// TIA Portal V16 export
// export: Created 2021-06-11T05:47:00.3145805Z, ExportSetting WithDefaults, DisplayName Totally Integrated Automation Portal, DisplayVersion V16 Update 4, DisplayName TIA Portal Version Control Interface, DisplayVersion V16 Update 2, DisplayName TIA Portal Openness, DisplayVersion V16 Update 4, DisplayName TIA Portal Teamcenter Gateway, DisplayVersion V16, DisplayName SINAMICS Startdrive Advanced, DisplayVersion V16 Update 5, DisplayName SINAMICS Startdrive G130, G150, S120, S150, SINAMICS MV, S210, DisplayVersion V16 Update 5, DisplayName SINAMICS Startdrive G110M, G120, G120C, G120D, G120P, G115D, DisplayVersion V16 Update 5, DisplayName STEP 7 Professional, DisplayVersion V16 Update 4, DisplayName SINUMERIK ONE STEP 7 Toolbox, DisplayVersion V16 Update 3, DisplayName STEP 7 Safety, DisplayVersion V16, DisplayName SINUMERIK 840D sl STEP 7 Toolbox, DisplayVersion V16 Update 2, DisplayName WinCC Advanced, DisplayVersion V16 Update 4
FUNCTION "FC_OperatingModes" : Void   // FC1601, LAD
{ S7_Optimized_Access := 'TRUE' }
VERSION : 0.1
// stored: AutoNumber false, IsIECCheckEnabled false, SetENOAutomatically true, UDAEnableTagReadback false
   VAR_TEMP
      tx_OperatingMode_KeyDisable : Bool;
      tb_DialogEnable : Byte;
      tx_DialogEnable : Array[0..7] of Bool;
      tint_Ret_Val : Int;
      WcsMcs_Edge : Bool;
      WcsMcs_Flag : Bool;
   END_VAR
BEGIN

REGION Network 1: MCP
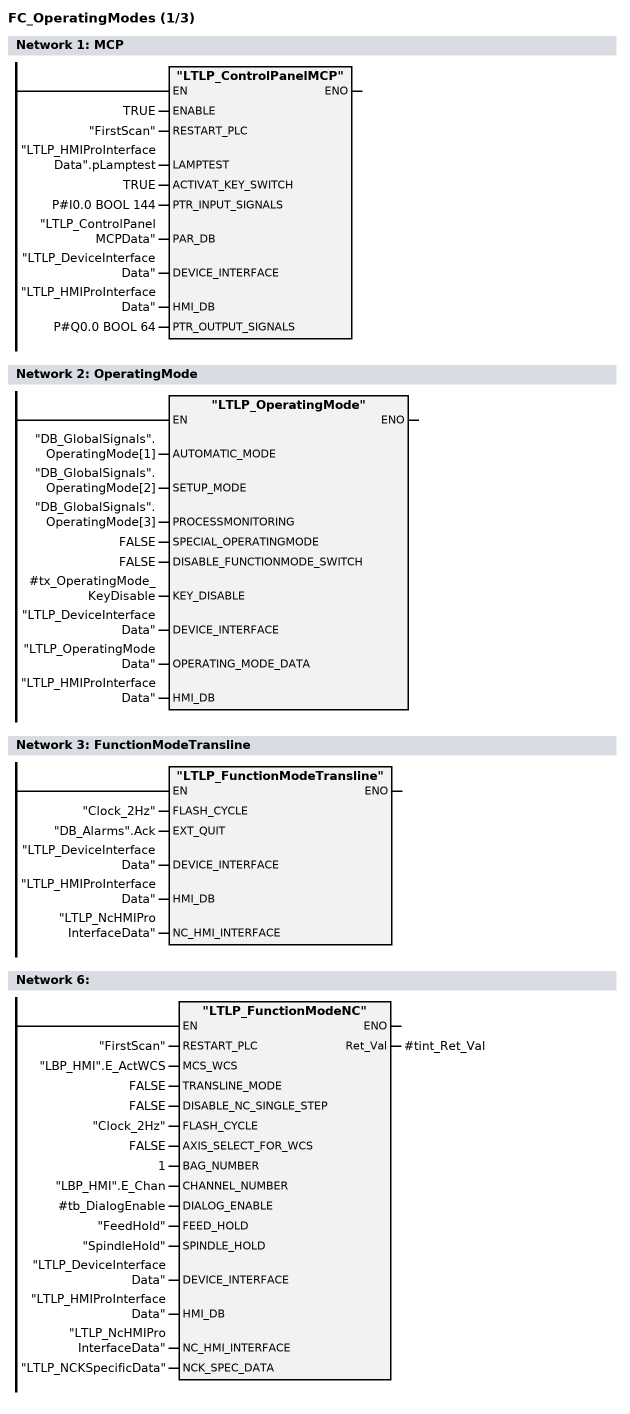
   RUNG wire#powerrail
      "LTLP_ControlPanelMCP"(ENABLE := TRUE, RESTART_PLC := "FirstScan", LAMPTEST := "LTLP_HMIProInterfaceData".pLamptest, ACTIVAT_KEY_SWITCH := TRUE, PTR_INPUT_SIGNALS := P#I0.0 BOOL 144, PAR_DB := "LTLP_ControlPanelMCPData", DEVICE_INTERFACE := "LTLP_DeviceInterfaceData", HMI_DB := "LTLP_HMIProInterfaceData", PTR_OUTPUT_SIGNALS := P#Q0.0 BOOL 64)
   END_RUNG
   // the same network as SCL:
   "LTLP_ControlPanelMCP"(ENABLE := TRUE,
                          RESTART_PLC := "FirstScan",
                          LAMPTEST := "LTLP_HMIProInterfaceData".pLamptest,
                          ACTIVAT_KEY_SWITCH := TRUE,
                          PTR_INPUT_SIGNALS := P#I0.0 BOOL 144,
                          PAR_DB := "LTLP_ControlPanelMCPData",
                          DEVICE_INTERFACE := "LTLP_DeviceInterfaceData",
                          HMI_DB := "LTLP_HMIProInterfaceData",
                          PTR_OUTPUT_SIGNALS := P#Q0.0 BOOL 64);
END_REGION

REGION Network 2: OperatingMode
   RUNG wire#powerrail
      "LTLP_OperatingMode"(AUTOMATIC_MODE := "DB_GlobalSignals".OperatingMode[1], SETUP_MODE := "DB_GlobalSignals".OperatingMode[2], PROCESSMONITORING := "DB_GlobalSignals".OperatingMode[3], SPECIAL_OPERATINGMODE := FALSE, DISABLE_FUNCTIONMODE_SWITCH := FALSE, KEY_DISABLE := #tx_OperatingMode_KeyDisable, DEVICE_INTERFACE := "LTLP_DeviceInterfaceData", OPERATING_MODE_DATA := "LTLP_OperatingModeData", HMI_DB := "LTLP_HMIProInterfaceData")
   END_RUNG
   // the same network as SCL:
   "LTLP_OperatingMode"(AUTOMATIC_MODE := "DB_GlobalSignals".OperatingMode[1],
                        SETUP_MODE := "DB_GlobalSignals".OperatingMode[2],
                        PROCESSMONITORING := "DB_GlobalSignals".OperatingMode[3],
                        SPECIAL_OPERATINGMODE := FALSE,
                        DISABLE_FUNCTIONMODE_SWITCH := FALSE,
                        KEY_DISABLE := #tx_OperatingMode_KeyDisable,
                        DEVICE_INTERFACE := "LTLP_DeviceInterfaceData",
                        OPERATING_MODE_DATA := "LTLP_OperatingModeData",
                        HMI_DB := "LTLP_HMIProInterfaceData");
END_REGION

REGION Network 3: FunctionModeTransline
   RUNG wire#powerrail
      "LTLP_FunctionModeTransline"(FLASH_CYCLE := "Clock_2Hz", EXT_QUIT := "DB_Alarms".Ack, DEVICE_INTERFACE := "LTLP_DeviceInterfaceData", HMI_DB := "LTLP_HMIProInterfaceData", NC_HMI_INTERFACE := "LTLP_NcHMIProInterfaceData")
   END_RUNG
   // the same network as SCL:
   "LTLP_FunctionModeTransline"(FLASH_CYCLE := "Clock_2Hz",
                           EXT_QUIT := "DB_Alarms".Ack,
                           DEVICE_INTERFACE := "LTLP_DeviceInterfaceData",
                           HMI_DB := "LTLP_HMIProInterfaceData",
                           NC_HMI_INTERFACE := "LTLP_NcHMIProInterfaceData");
END_REGION

REGION Network 4 (SCL)
   #tx_DialogEnable[0] := TRUE;
   #tx_DialogEnable[1] := TRUE;
   #tx_DialogEnable[2] := TRUE;
   #tx_DialogEnable[3] := FALSE;
   #tx_DialogEnable[4] := FALSE;
   #tx_DialogEnable[5] := FALSE;
   #tx_DialogEnable[6] := FALSE;
   #tx_DialogEnable[7] := TRUE;

   GATHER(IN := #tx_DialogEnable,
          OUT => #tb_DialogEnable);

   "LTLP_NCKSpecificData".Common.maxBAG := "LBP_ConfigData".MaxModeGroup;
   "LTLP_NCKSpecificData".Common.maxChannels := "LBP_ConfigData".MaxChan;
   "LTLP_NCKSpecificData".Common.maxAxis := "LBP_ConfigData".MaxAxis;

   "LTLP_NCKSpecificData".NCK.A_incInModeGroup := "LBP_NC".A_IncInModeGroup;
   "LTLP_NCKSpecificData".MMC.activeChannel := "LBP_HMI".E_Chan;

   //Flanke - System betriebsbereit
   "IDB_R_TRIG_SystemReady"(CLK := "LBP_NC".E_NCKready AND "LBP_NC".E_NCready AND "LBP_NC".E_DrivesInCylOp);

   //FeedStart im Hochlauf setzen
   IF "IDB_R_TRIG_SystemReady".Q THEN
       "LTLP_DeviceInterfaceData".inputs.mcpFunctions.feedStart := TRUE;
   ELSIF NOT "FeedHold" THEN
       "LTLP_DeviceInterfaceData".inputs.mcpFunctions.feedStart := FALSE;
   END_IF;
   //SpindleStart im Hochlauf setzen
   IF "IDB_R_TRIG_SystemReady".Q THEN
       "LTLP_DeviceInterfaceData".inputs.mcpFunctions.spindleStart := TRUE;
   ELSIF NOT "SpindleHold" THEN
       "LTLP_DeviceInterfaceData".inputs.mcpFunctions.spindleStart := FALSE;
   END_IF;
END_REGION

REGION Network 5 (SCL): bagDataSpecification
   // BAG
   "LTLP_NcHMIProInterfaceData".bagDataFeedback.auto := "LBP_ModeGroup".E_AUTO;
   "LTLP_NcHMIProInterfaceData".bagDataFeedback.mda := "LBP_ModeGroup".E_MDA;
   "LTLP_NcHMIProInterfaceData".bagDataFeedback.jog := "LBP_ModeGroup".E_JOG;
   "LTLP_NcHMIProInterfaceData".bagDataFeedback.inrement1 := "LBP_ModeGroup".E_INC1;
   "LTLP_NcHMIProInterfaceData".bagDataFeedback.inrement10 := "LBP_ModeGroup".E_INC10;
   "LTLP_NcHMIProInterfaceData".bagDataFeedback.inrement100 := "LBP_ModeGroup".E_INC100;
   "LTLP_NcHMIProInterfaceData".bagDataFeedback.increment1000 := "LBP_ModeGroup".E_INC1000;
   "LTLP_NcHMIProInterfaceData".bagDataFeedback.increment10000 := "LBP_ModeGroup".E_INC10000;
   "LTLP_NcHMIProInterfaceData".bagDataFeedback.incremetVariable := "LBP_ModeGroup".E_INCVar;
   "LTLP_NcHMIProInterfaceData".bagDataFeedback.gotoRefPoint := "LBP_ModeGroup".E_REF;
   "LTLP_NcHMIProInterfaceData".bagDataFeedback.teach := "LBP_ModeGroup".E_TEACHIN;

   // Channel
   "LTLP_NcHMIProInterfaceData".channelDataFeedback.rapidTraverse := "LTLP_DeviceInterfaceData".inputs.mcpFunctions.rapid;
   "LTLP_NcHMIProInterfaceData".channelDataFeedback.motionPlus := "LTLP_DeviceInterfaceData".inputs.mcpFunctions.motionPlus;
   "LTLP_NcHMIProInterfaceData".channelDataFeedback.motionMinus := "LTLP_DeviceInterfaceData".inputs.mcpFunctions.motionMinus;
   "LTLP_NcHMIProInterfaceData".channelDataFeedback.ncStart := "LTLP_DeviceInterfaceData".inputs.mcpFunctions.ncStart;
   "LTLP_NcHMIProInterfaceData".channelDataFeedback.ncStop := "LTLP_DeviceInterfaceData".inputs.mcpFunctions.ncStop;
   "LTLP_NcHMIProInterfaceData".channelDataFeedback.reset := "LTLP_DeviceInterfaceData".inputs.mcpFunctions.reset;
   "LTLP_NcHMIProInterfaceData".channelDataFeedback.singleBlock := "LBP_Chan1".A_SBL;

   // Axis
   "LTLP_NcHMIProInterfaceData".axisFeedback.rapidTraverse := "LTLP_DeviceInterfaceData".inputs.mcpFunctions.rapid;
   "LTLP_NcHMIProInterfaceData".axisFeedback.motionPlus := "LTLP_DeviceInterfaceData".inputs.mcpFunctions.motionPlus;
   "LTLP_NcHMIProInterfaceData".axisFeedback.motionMinus := "LTLP_DeviceInterfaceData".inputs.mcpFunctions.motionMinus;

   // Achse abwählen, falls AUTO oder MDA aktiv
   IF "LTLP_NcHMIProInterfaceData".bagDataFeedback.auto OR "LTLP_NcHMIProInterfaceData".bagDataFeedback.mda THEN
       "LTLP_NcHMIProInterfaceData".fromPlc.axisNoMcp := 0;
   END_IF;
END_REGION

REGION Network 6
   RUNG wire#powerrail
      "LTLP_FunctionModeNC"(RESTART_PLC := "FirstScan", MCS_WCS := "LBP_HMI".E_ActWCS, TRANSLINE_MODE := FALSE, DISABLE_NC_SINGLE_STEP := FALSE, FLASH_CYCLE := "Clock_2Hz", AXIS_SELECT_FOR_WCS := FALSE, BAG_NUMBER := 1, CHANNEL_NUMBER := "LBP_HMI".E_Chan, DIALOG_ENABLE := #tb_DialogEnable, FEED_HOLD := "FeedHold", SPINDLE_HOLD := "SpindleHold", DEVICE_INTERFACE := "LTLP_DeviceInterfaceData", HMI_DB := "LTLP_HMIProInterfaceData", NC_HMI_INTERFACE := "LTLP_NcHMIProInterfaceData", NCK_SPEC_DATA := "LTLP_NCKSpecificData", Ret_Val => #tint_Ret_Val)
   END_RUNG
   // the same network as SCL:
   #tint_Ret_Val := "LTLP_FunctionModeNC"(RESTART_PLC := "FirstScan",
                           MCS_WCS := "LBP_HMI".E_ActWCS,
                           TRANSLINE_MODE := FALSE,
                           DISABLE_NC_SINGLE_STEP := FALSE,
                           FLASH_CYCLE := "Clock_2Hz",
                           AXIS_SELECT_FOR_WCS := FALSE,
                           BAG_NUMBER := 1,
                           CHANNEL_NUMBER := "LBP_HMI".E_Chan,
                           DIALOG_ENABLE := #tb_DialogEnable,
                           FEED_HOLD := "FeedHold",
                           SPINDLE_HOLD := "SpindleHold",
                           DEVICE_INTERFACE := "LTLP_DeviceInterfaceData",
                           HMI_DB := "LTLP_HMIProInterfaceData",
                           NC_HMI_INTERFACE := "LTLP_NcHMIProInterfaceData",
                           NCK_SPEC_DATA := "LTLP_NCKSpecificData");
END_REGION

REGION Network 7: Betriebsarten
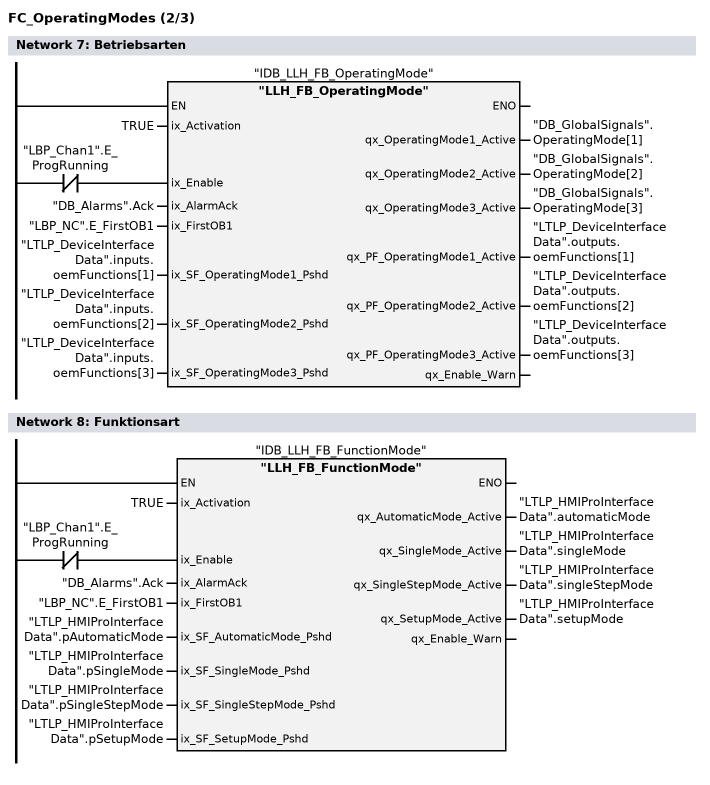
   RUNG wire#powerrail
      "IDB_LLH_FB_OperatingMode"(ix_Enable := wire#w1, ix_Activation := TRUE, ix_AlarmAck := "DB_Alarms".Ack, ix_FirstOB1 := "LBP_NC".E_FirstOB1, ix_SF_OperatingMode1_Pshd := "LTLP_DeviceInterfaceData".inputs.oemFunctions[1], ix_SF_OperatingMode2_Pshd := "LTLP_DeviceInterfaceData".inputs.oemFunctions[2], ix_SF_OperatingMode3_Pshd := "LTLP_DeviceInterfaceData".inputs.oemFunctions[3], qx_OperatingMode1_Active => "DB_GlobalSignals".OperatingMode[1], qx_OperatingMode2_Active => "DB_GlobalSignals".OperatingMode[2], qx_OperatingMode3_Active => "DB_GlobalSignals".OperatingMode[3], qx_PF_OperatingMode1_Active => "LTLP_DeviceInterfaceData".outputs.oemFunctions[1], qx_PF_OperatingMode2_Active => "LTLP_DeviceInterfaceData".outputs.oemFunctions[2], qx_PF_OperatingMode3_Active => "LTLP_DeviceInterfaceData".outputs.oemFunctions[3], qx_Enable_Warn =>)
   END_RUNG
   RUNG wire#powerrail
      I_Contact( "LBP_Chan1".E_ProgRunning )
   END_RUNG wire#w1
   // the same network as SCL:
   "IDB_LLH_FB_OperatingMode"(ix_Activation := TRUE,   // "LLH_FB_OperatingMode"
                           ix_Enable := NOT "LBP_Chan1".E_ProgRunning,
                           ix_AlarmAck := "DB_Alarms".Ack,
                           ix_FirstOB1 := "LBP_NC".E_FirstOB1,
                           ix_SF_OperatingMode1_Pshd := "LTLP_DeviceInterfaceData".inputs.oemFunctions[1],
                           ix_SF_OperatingMode2_Pshd := "LTLP_DeviceInterfaceData".inputs.oemFunctions[2],
                           ix_SF_OperatingMode3_Pshd := "LTLP_DeviceInterfaceData".inputs.oemFunctions[3],
                           qx_OperatingMode1_Active => "DB_GlobalSignals".OperatingMode[1],
                           qx_OperatingMode2_Active => "DB_GlobalSignals".OperatingMode[2],
                           qx_OperatingMode3_Active => "DB_GlobalSignals".OperatingMode[3],
                           qx_PF_OperatingMode1_Active => "LTLP_DeviceInterfaceData".outputs.oemFunctions[1],
                           qx_PF_OperatingMode2_Active => "LTLP_DeviceInterfaceData".outputs.oemFunctions[2],
                           qx_PF_OperatingMode3_Active => "LTLP_DeviceInterfaceData".outputs.oemFunctions[3]);
END_REGION

REGION Network 8: Funktionsart
   RUNG wire#powerrail
      "IDB_LLH_FB_FunctionMode"(ix_Enable := wire#w1, ix_Activation := TRUE, ix_AlarmAck := "DB_Alarms".Ack, ix_FirstOB1 := "LBP_NC".E_FirstOB1, ix_SF_AutomaticMode_Pshd := "LTLP_HMIProInterfaceData".pAutomaticMode, ix_SF_SingleMode_Pshd := "LTLP_HMIProInterfaceData".pSingleMode, ix_SF_SingleStepMode_Pshd := "LTLP_HMIProInterfaceData".pSingleStepMode, ix_SF_SetupMode_Pshd := "LTLP_HMIProInterfaceData".pSetupMode, qx_AutomaticMode_Active => "LTLP_HMIProInterfaceData".automaticMode, qx_SingleMode_Active => "LTLP_HMIProInterfaceData".singleMode, qx_SingleStepMode_Active => "LTLP_HMIProInterfaceData".singleStepMode, qx_SetupMode_Active => "LTLP_HMIProInterfaceData".setupMode, qx_Enable_Warn =>)
   END_RUNG
   RUNG wire#powerrail
      I_Contact( "LBP_Chan1".E_ProgRunning )
   END_RUNG wire#w1
   // the same network as SCL:
   "IDB_LLH_FB_FunctionMode"(ix_Activation := TRUE,   // "LLH_FB_FunctionMode"
                           ix_Enable := NOT "LBP_Chan1".E_ProgRunning,
                           ix_AlarmAck := "DB_Alarms".Ack,
                           ix_FirstOB1 := "LBP_NC".E_FirstOB1,
                           ix_SF_AutomaticMode_Pshd := "LTLP_HMIProInterfaceData".pAutomaticMode,
                           ix_SF_SingleMode_Pshd := "LTLP_HMIProInterfaceData".pSingleMode,
                           ix_SF_SingleStepMode_Pshd := "LTLP_HMIProInterfaceData".pSingleStepMode,
                           ix_SF_SetupMode_Pshd := "LTLP_HMIProInterfaceData".pSetupMode,
                           qx_AutomaticMode_Active => "LTLP_HMIProInterfaceData".automaticMode,
                           qx_SingleMode_Active => "LTLP_HMIProInterfaceData".singleMode,
                           qx_SingleStepMode_Active => "LTLP_HMIProInterfaceData".singleStepMode,
                           qx_SetupMode_Active => "LTLP_HMIProInterfaceData".setupMode);
END_REGION

REGION Network 9: ModeGroup
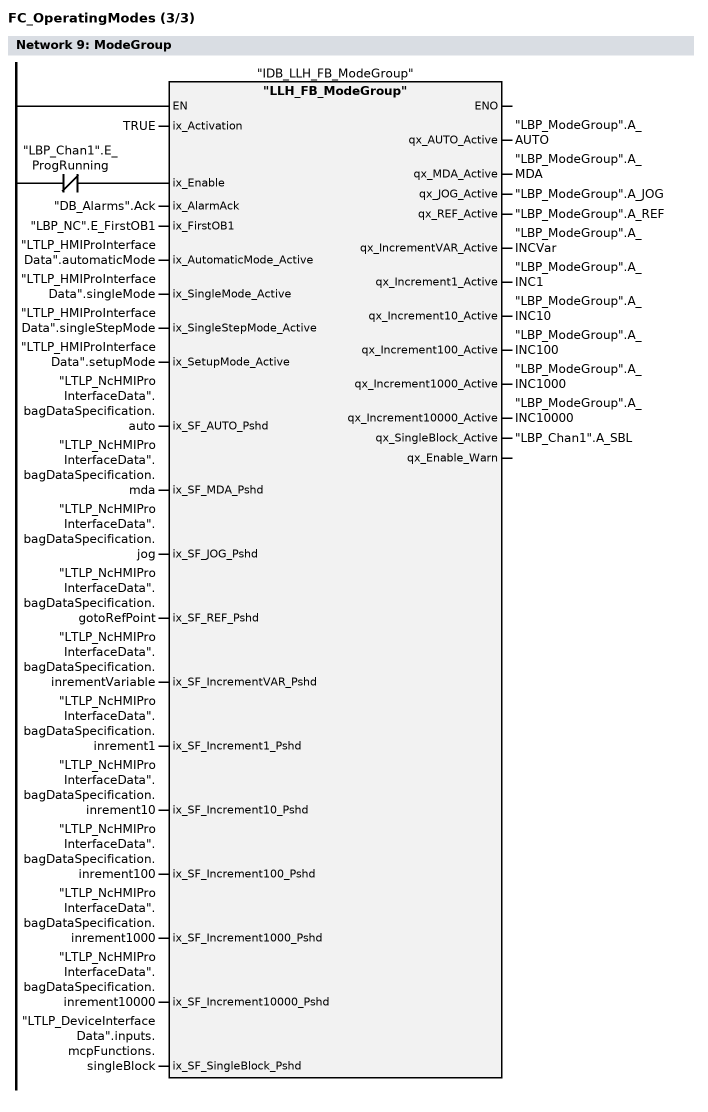
   RUNG wire#powerrail
      "IDB_LLH_FB_ModeGroup"(ix_Enable := wire#w1, ix_Activation := TRUE, ix_AlarmAck := "DB_Alarms".Ack, ix_FirstOB1 := "LBP_NC".E_FirstOB1, ix_AutomaticMode_Active := "LTLP_HMIProInterfaceData".automaticMode, ix_SingleMode_Active := "LTLP_HMIProInterfaceData".singleMode, ix_SingleStepMode_Active := "LTLP_HMIProInterfaceData".singleStepMode, ix_SetupMode_Active := "LTLP_HMIProInterfaceData".setupMode, ix_SF_AUTO_Pshd := "LTLP_NcHMIProInterfaceData".bagDataSpecification.auto, ix_SF_MDA_Pshd := "LTLP_NcHMIProInterfaceData".bagDataSpecification.mda, ix_SF_JOG_Pshd := "LTLP_NcHMIProInterfaceData".bagDataSpecification.jog, ix_SF_REF_Pshd := "LTLP_NcHMIProInterfaceData".bagDataSpecification.gotoRefPoint, ix_SF_IncrementVAR_Pshd := "LTLP_NcHMIProInterfaceData".bagDataSpecification.inrementVariable, ix_SF_Increment1_Pshd := "LTLP_NcHMIProInterfaceData".bagDataSpecification.inrement1, ix_SF_Increment10_Pshd := "LTLP_NcHMIProInterfaceData".bagDataSpecification.inrement10, ix_SF_Increment100_Pshd := "LTLP_NcHMIProInterfaceData".bagDataSpecification.inrement100, ix_SF_Increment1000_Pshd := "LTLP_NcHMIProInterfaceData".bagDataSpecification.inrement1000, ix_SF_Increment10000_Pshd := "LTLP_NcHMIProInterfaceData".bagDataSpecification.inrement10000, ix_SF_SingleBlock_Pshd := "LTLP_DeviceInterfaceData".inputs.mcpFunctions.singleBlock, qx_AUTO_Active => "LBP_ModeGroup".A_AUTO, qx_MDA_Active => "LBP_ModeGroup".A_MDA, qx_JOG_Active => "LBP_ModeGroup".A_JOG, qx_REF_Active => "LBP_ModeGroup".A_REF, qx_IncrementVAR_Active => "LBP_ModeGroup".A_INCVar, qx_Increment1_Active => "LBP_ModeGroup".A_INC1, qx_Increment10_Active => "LBP_ModeGroup".A_INC10, qx_Increment100_Active => "LBP_ModeGroup".A_INC100, qx_Increment1000_Active => "LBP_ModeGroup".A_INC1000, qx_Increment10000_Active => "LBP_ModeGroup".A_INC10000, qx_SingleBlock_Active => "LBP_Chan1".A_SBL, qx_Enable_Warn =>)
   END_RUNG
   RUNG wire#powerrail
      I_Contact( "LBP_Chan1".E_ProgRunning )
   END_RUNG wire#w1
   // the same network as SCL:
   "IDB_LLH_FB_ModeGroup"(ix_Activation := TRUE,   // "LLH_FB_ModeGroup"
                          ix_Enable := NOT "LBP_Chan1".E_ProgRunning,
                          ix_AlarmAck := "DB_Alarms".Ack,
                          ix_FirstOB1 := "LBP_NC".E_FirstOB1,
                          ix_AutomaticMode_Active := "LTLP_HMIProInterfaceData".automaticMode,
                          ix_SingleMode_Active := "LTLP_HMIProInterfaceData".singleMode,
                          ix_SingleStepMode_Active := "LTLP_HMIProInterfaceData".singleStepMode,
                          ix_SetupMode_Active := "LTLP_HMIProInterfaceData".setupMode,
                          ix_SF_AUTO_Pshd := "LTLP_NcHMIProInterfaceData".bagDataSpecification.auto,
                          ix_SF_MDA_Pshd := "LTLP_NcHMIProInterfaceData".bagDataSpecification.mda,
                          ix_SF_JOG_Pshd := "LTLP_NcHMIProInterfaceData".bagDataSpecification.jog,
                          ix_SF_REF_Pshd := "LTLP_NcHMIProInterfaceData".bagDataSpecification.gotoRefPoint,
                          ix_SF_IncrementVAR_Pshd := "LTLP_NcHMIProInterfaceData".bagDataSpecification.inrementVariable,
                          ix_SF_Increment1_Pshd := "LTLP_NcHMIProInterfaceData".bagDataSpecification.inrement1,
                          ix_SF_Increment10_Pshd := "LTLP_NcHMIProInterfaceData".bagDataSpecification.inrement10,
                          ix_SF_Increment100_Pshd := "LTLP_NcHMIProInterfaceData".bagDataSpecification.inrement100,
                          ix_SF_Increment1000_Pshd := "LTLP_NcHMIProInterfaceData".bagDataSpecification.inrement1000,
                          ix_SF_Increment10000_Pshd := "LTLP_NcHMIProInterfaceData".bagDataSpecification.inrement10000,
                          ix_SF_SingleBlock_Pshd := "LTLP_DeviceInterfaceData".inputs.mcpFunctions.singleBlock,
                          qx_AUTO_Active => "LBP_ModeGroup".A_AUTO,
                          qx_MDA_Active => "LBP_ModeGroup".A_MDA,
                          qx_JOG_Active => "LBP_ModeGroup".A_JOG,
                          qx_REF_Active => "LBP_ModeGroup".A_REF,
                          qx_IncrementVAR_Active => "LBP_ModeGroup".A_INCVar,
                          qx_Increment1_Active => "LBP_ModeGroup".A_INC1,
                          qx_Increment10_Active => "LBP_ModeGroup".A_INC10,
                          qx_Increment100_Active => "LBP_ModeGroup".A_INC100,
                          qx_Increment1000_Active => "LBP_ModeGroup".A_INC1000,
                          qx_Increment10000_Active => "LBP_ModeGroup".A_INC10000,
                          qx_SingleBlock_Active => "LBP_Chan1".A_SBL);
END_REGION

REGION Network 10 (SCL): HMI - MKS/WKS-Anzeige
   // Positive Flanke
   #WcsMcs_Edge := "LBP_HMI".E_ActWCS AND NOT #WcsMcs_Flag;
   // Flankenauswertung - Hilfsvariable
   #WcsMcs_Flag := "LBP_HMI".E_ActWCS;
   // Anzeige umschalten
   "LBP_HMI".A_ActWCS := ("LBP_HMI".A_ActWCS XOR #WcsMcs_Edge);
END_REGION
END_FUNCTION
